# EPICS substitutions: ct-eps/csx-epsApp/Db/ct-eps-plc-misc.substitutions
file ct-eps-plc-misc.template
{
	pattern {Sys, PLC}
			{XF:23ID-CT, XF_23ID_EPS_ES1_PLC_F1}
}
